{attribute addProperty BoxType "EJ6910-0000-0018"}
{attribute addProperty Id "FSLOGIC_InputsAT %I*FSLOGIC_Inputs_8BA5C9331620FSLOGIC_OutputsAT %Q*EMPTY_STRUCTURE000WcStateAT %I*WcState_98A4DF7520.250InfoDataAT %I*InfoData_BC63D37F80100"}
{attribute addProperty CRC "1002942579"}
{attribute addProperty SizeInBites "98"}
{attribute addProperty SizeInBytes "12.25"}
TYPE EJ6910_4EA245C6 :
STRUCT
	{attribute addProperty Name "FSLOGIC_Inputs"}
	FSLOGIC_Inputs : FSLOGIC_Inputs_8BA5C933;
	{attribute addProperty Name "FSLOGIC_Outputs"}
	FSLOGIC_Outputs : EMPTY_STRUCTURE;
	{attribute addProperty Name "WcState"}
	WcState : WcState_98A4DF75;
	{attribute addProperty Name "InfoData"}
	InfoData : InfoData_BC63D37F;
END_STRUCT
END_TYPE

(* stored: Version 1.2.0.0, ProductVersion 3.1.4024.9
   DUT EJ6910_4EA245C6: Id {80b4eba5-ca61-470c-afdc-a0e85d4a8d40} *)
